FUNCTION_BLOCK LOADL (* Local channel publisher for workpiece loading *)
  (* Standard: 61499-2; Classification: Simulation *)
  (* Version 0.1, 2004-10-23, JHC, Rockwell Automation, Added default ID value. *)
  (* Version 0.0, 2004-10-08, JHC, Rockwell Automation *)
  (* Compiler header: package fb.rt.mva; import fb.rt.net.*; *)
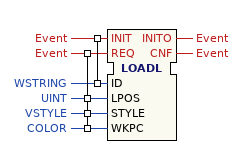
  EVENT_INPUT
    INIT WITH ID; (* Service Initialization *)
    REQ WITH LPOS, STYLE, WKPC; (* Publish LOAD command *)
  END_EVENT
  EVENT_OUTPUT
    INITO; (* Initialization Confirm *)
    CNF; (* Execution Confirmation *)
  END_EVENT
  VAR_INPUT
    ID : WSTRING; (* Local Group ID, default = FB instance name *)
    LPOS : UINT; (* Load Position in % of Conveyor Length *)
    STYLE : VSTYLE := NONE; (* Input Workpiece style *)
    WKPC : COLOR := yellow; (* Input Workpiece Color *)
  END_VAR
  FBS
    PUB : PUBL_3;
  END_FBS
  EVENT_CONNECTIONS
    INIT TO PUB.INIT;
    REQ TO PUB.REQ;
    PUB.INITO TO INITO;
    PUB.CNF TO CNF;
  END_CONNECTIONS
  DATA_CONNECTIONS
    ID TO PUB.ID;
    LPOS TO PUB.SD_1;
    STYLE TO PUB.SD_2;
    WKPC TO PUB.SD_3;
  END_CONNECTIONS
END_FUNCTION_BLOCK
